// TIA Portal project "practica kp8" (V15)

(* hardware
DEVICE "S7-1200 station_1"  S7-1200 Station
   slot 0: "Rack_0"  S7-1200 Rack  Rack  V1.0
   slot 1: "PLC_1"  CPU 1214C AC/DC/Rly  6ES7 214-1BE30-0XB0  V2.2
   slot 3: "AQ 1x12BIT_1"  AQ1 signal board  6ES7 232-4HA30-0XB0  V1.0
DEVICE "KP8_1"  SIMATIC Key Panel
   slot 0: "Rack"  Rail  V1.0
   slot 0: "KP8_1"  KP8  6AV3 688-3AY36-0AX0  R01.00.00
*)

// ===== PLC "PLC_1"  CPU 1214C AC/DC/Rly =====

VAR_GLOBAL   // PLC tag table "Tabla de variables estándar"
   "botón" AT %I2.7 : Bool;
   "color rojo" AT %Q2.7 : Bool;
   "Tag_3" AT %M40.0 : Bool;
   "color verde" AT %Q3.7 : Bool;
END_VAR

ORGANIZATION_BLOCK "Main"   // OB1, LAD, ProgramCycle
TITLE = "Main Program Sweep (Cycle)"
{ S7_Optimized_Access := 'TRUE' }
VERSION : 0.1
   VAR_TEMP   // added for the SCL form of the ladder/FBD networks
      _w1 : Bool;
      _w2 : Bool;
      _w3 : Bool;
   END_VAR
BEGIN

REGION Network 1
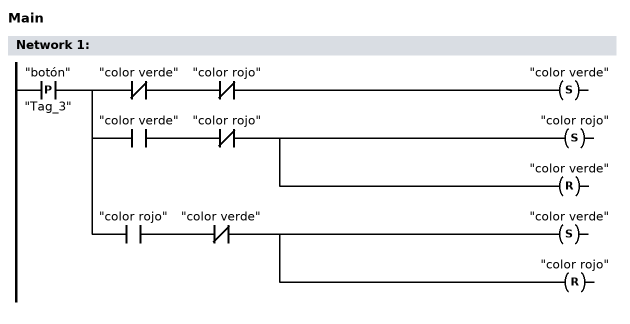
   RUNG wire#powerrail
      P_Contact(operand := "botón", bit := "Tag_3")
      wire#w1
      I_Contact( "color verde" )
      I_Contact( "color rojo" )
      S_Coil( "color verde" )
   END_RUNG
   RUNG wire#w1
      Contact( "color verde" )
      I_Contact( "color rojo" )
      wire#w2
      S_Coil( "color rojo" )
   END_RUNG
   RUNG wire#w2
      R_Coil( "color verde" )
   END_RUNG
   RUNG wire#w1
      Contact( "color rojo" )
      I_Contact( "color verde" )
      wire#w3
      S_Coil( "color verde" )
   END_RUNG
   RUNG wire#w3
      R_Coil( "color rojo" )
   END_RUNG
   // the same network as SCL:
   #_w1 := "botón" AND NOT "Tag_3";   // rising edge of "botón"
   "Tag_3" := "botón";
   IF #_w1 AND NOT "color verde" AND NOT "color rojo" THEN "color verde" := TRUE; END_IF;
   #_w2 := #_w1 AND "color verde" AND NOT "color rojo";
   IF #_w2 THEN
       "color rojo" := TRUE;
       "color verde" := FALSE;
   END_IF;
   #_w3 := #_w1 AND "color rojo" AND NOT "color verde";
   IF #_w3 THEN
       "color verde" := TRUE;
       "color rojo" := FALSE;
   END_IF;
END_REGION
END_ORGANIZATION_BLOCK